FUNCTION FUN_GetNeedleCoordinates : BOOL
VAR_INPUT
	uiLocation		: UINT	; // 0 : From RoundBelt , 1 :From Turn table
	uiBox			: UINT ; // 0 or 1 
	uiClip			: INT ; // 0~3
	uiNeedleLocation : INT ; // 0~49
END_VAR

VAR_OUTPUT
	NeedleCoordinate		: st_Coordinate;
END_VAR

VAR
	BasePos 			: st_Coordinate;
	NeedlePosition		: st_Coordinate		;
	NeedleColumns : INT;
    NeedliRows    : INT;
	bDataCheck			 : BOOL;
	bGetPositionDone	:BOOL;
	PositionTable		:ST_PositionTable;
	i : INT;
END_VAR

IF (uiLocation =0 OR uiLocation = 1 ) AND (uiBox =0 OR uiBox =1) AND (uiClip>=0 AND uiClip <=3) AND (uiNeedleLocation >=0 AND uiNeedleLocation <=49) THEN
		bDataCheck := TRUE;
	ELSE
		bDataCheck := FALSE;
		FUN_GetNeedleCoordinates:=FALSE;
END_IF //Check data is valid

IF bDataCheck THEN
	
	CASE uiLocation OF	
		
	0:
	FOR i:=1 TO 200 BY 1 DO
 		IF 		DAS_CoreSys.MachineControl.CurrentData.PositionTable[i].Clip =UINT_TO_INT(uiClip) 
			AND DAS_CoreSys.MachineControl.CurrentData.PositionTable[i].Index= uiBox +1
			AND DAS_CoreSys.MachineControl.CurrentData.PositionTable[i].Zone ='Q' THEN
				PositionTable := DAS_CoreSys.MachineControl.CurrentData.PositionTable[i];
				EXIT;
		END_IF
		bGetPositionDone:=FALSE;
	END_FOR
	BasePos.X  :=  PositionTable.X_Pos;
	BasePos.Y   :=  PositionTable.Y_Pos;

	NeedleColumns := DINT_TO_INT(TRUNC(uiNeedleLocation / 10.0));
	NeedliRows    := LREAL_TO_INT(uiNeedleLocation MOD 10);

	NeedlePosition.Y := BasePos.Y + (DAS_CoreSys.MachineControl.CurrentData.Mechanical.Allocate_box_leftandRight_Distance * NeedleColumns);
	NeedlePosition.X := BasePos.X - (DAS_CoreSys.MachineControl.CurrentData.Mechanical.Allocate_box_UpandDown_Distance * NeedliRows);
	NeedleCoordinate:=NeedlePosition;
	bGetPositionDone:=TRUE;
	
1:
	
	FOR i:=1 TO 200 BY 1 DO
 		IF 		DAS_CoreSys.MachineControl.CurrentData.PositionTable[i].Clip = UINT_TO_INT(uiClip) 
			AND DAS_CoreSys.MachineControl.CurrentData.PositionTable[i].Index= uiBox +1
			AND DAS_CoreSys.MachineControl.CurrentData.PositionTable[i].Zone ='T' THEN
				PositionTable := DAS_CoreSys.MachineControl.CurrentData.PositionTable[i];
				EXIT;
		END_IF
		bGetPositionDone:=FALSE;
	END_FOR
	BasePos.X  :=  PositionTable.X_Pos;
	BasePos.Y   :=  PositionTable.Y_Pos;

	NeedleColumns := DINT_TO_INT(TRUNC(uiNeedleLocation / 10.0));
	NeedliRows    := LREAL_TO_INT(uiNeedleLocation MOD 10);

	NeedlePosition.Y := BasePos.Y + (DAS_CoreSys.MachineControl.CurrentData.Mechanical.Allocate_box_leftandRight_Distance * NeedleColumns);
	NeedlePosition.X := BasePos.X - (DAS_CoreSys.MachineControl.CurrentData.Mechanical.Allocate_box_UpandDown_Distance * NeedliRows);
	NeedleCoordinate:=NeedlePosition;
	bGetPositionDone:=TRUE;
	
	
	ELSE
		bGetPositionDone:=FALSE;	//Should not happen
 END_CASE
END_IF

FUN_GetNeedleCoordinates:=bGetPositionDone;

END_FUNCTION

(* stored: Version 1.1.0.1, ProductVersion 3.1.4024.13
   POU FUN_GetNeedleCoordinates: Id {720f16c8-389f-48fc-88b7-eee45b9714be}, SpecialFunc None *)
